// TIA Portal V20 export
FUNCTION "V103" : Void   // FC5, FBD
{ S7_Optimized_Access := 'TRUE' }
// stored: SetENOAutomatically false
   VAR_TEMP
      Temp : "DigVal";
      Temp_1 : "DigVal";
      State : "Service_States";
   END_VAR
BEGIN

REGION Network 1: Channel input
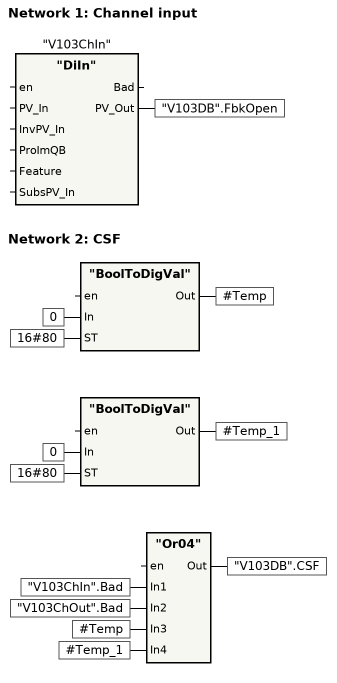
   "V103ChIn"(PV_Out => "V103DB".FbkOpen);   // "DiIn"
END_REGION

REGION Network 2: CSF
   "BoolToDigVal"(In := 0, ST := 16#80, Out => #Temp);
   "BoolToDigVal"(In := 0, ST := 16#80, Out => #Temp_1);
   "Or04"(In1 := "V103ChIn".Bad, In2 := "V103ChOut".Bad, In3 := #Temp, In4 := #Temp_1, Out => "V103DB".CSF);
END_REGION

REGION Network 3: VlvAn Intlock
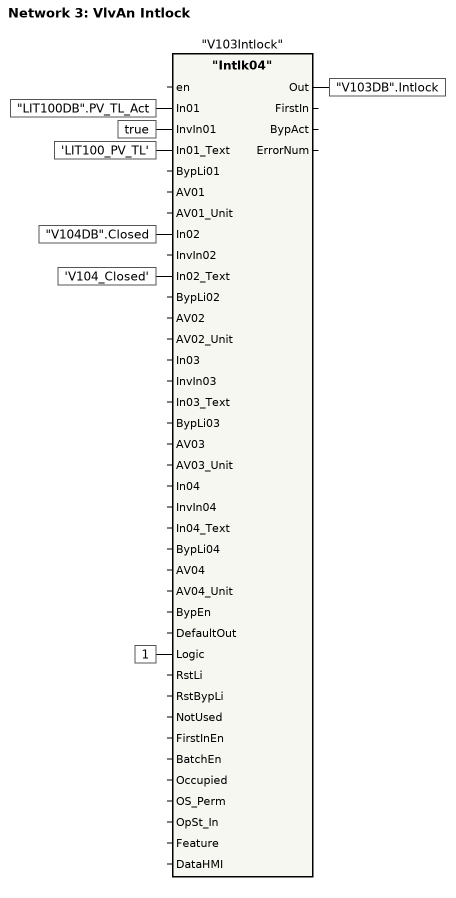
   "V103Intlock"(In01 := "LIT100DB".PV_TL_Act,   // "Intlk04"
                 InvIn01 := true,
                 In01_Text := 'LIT100_PV_TL',
                 In02 := "V104DB".Closed,
                 In02_Text := 'V104_Closed',
                 Logic := 1,
                 Out => "V103DB".Intlock);
END_REGION

REGION Network 4: VlvAnL
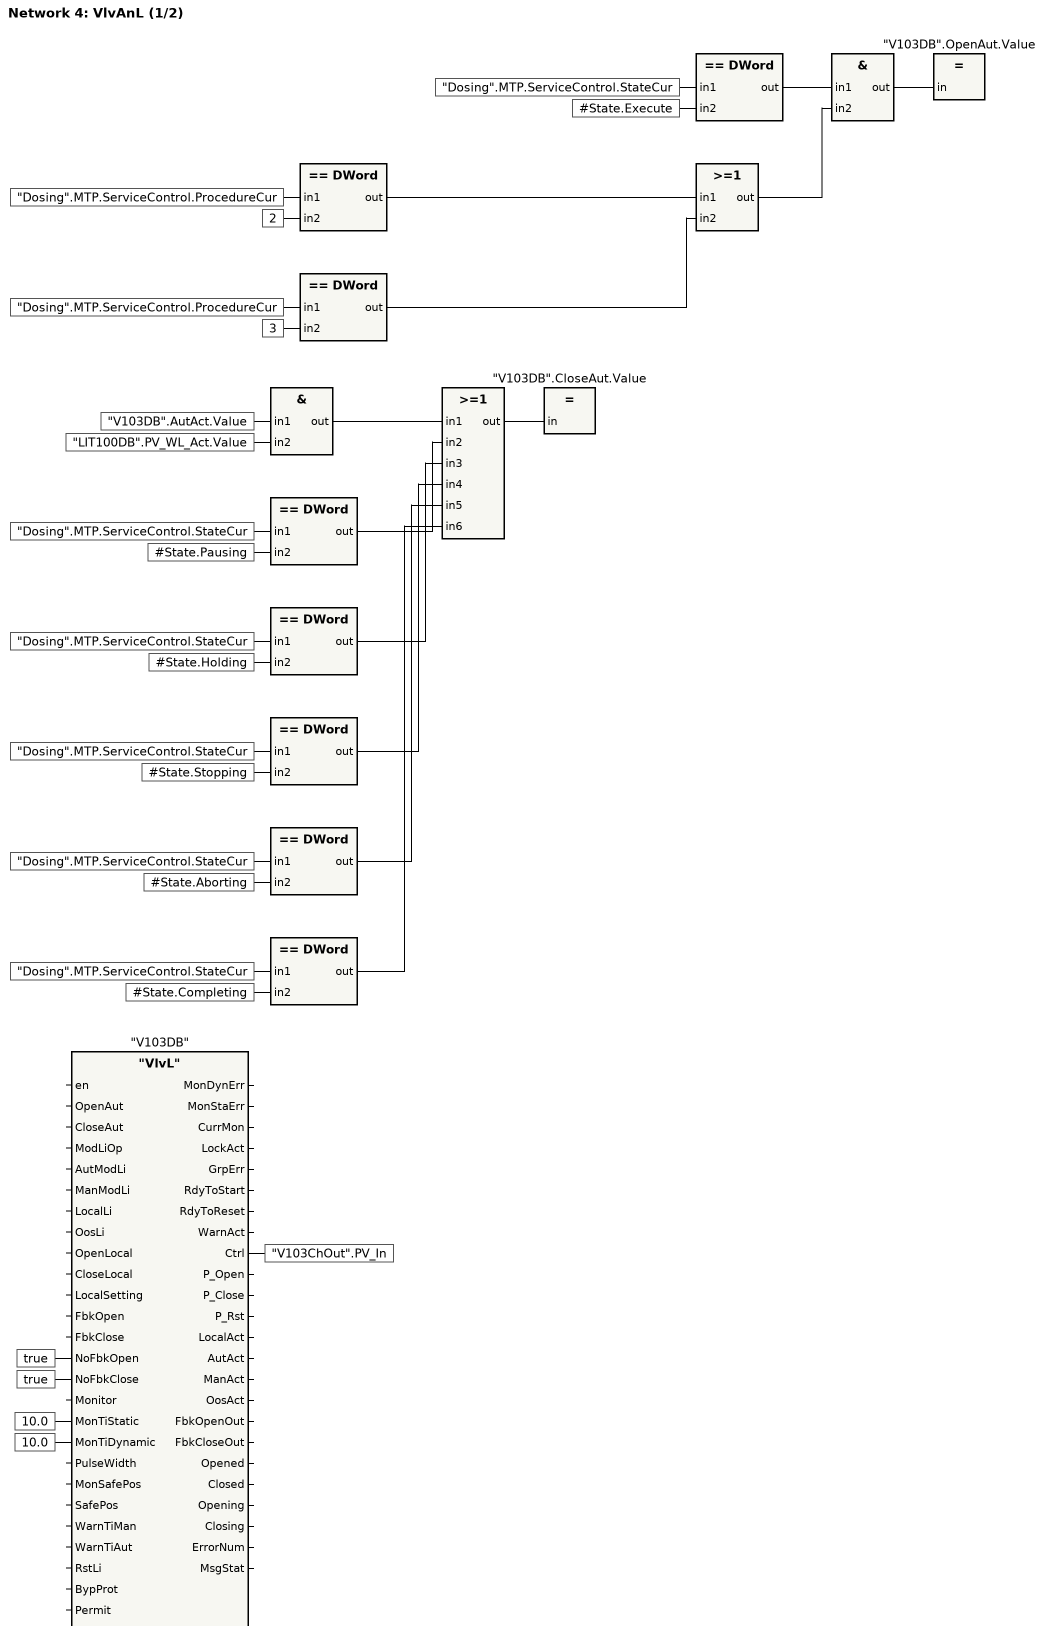
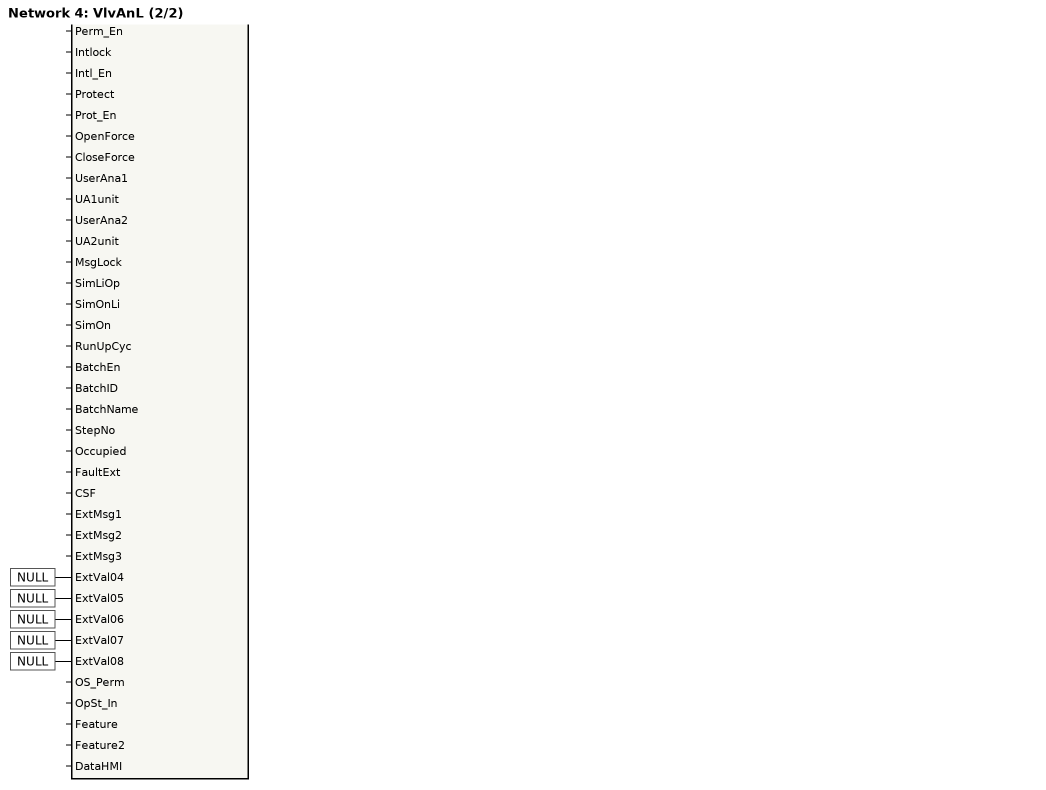
   "V103DB".OpenAut.Value := ("Dosing".MTP.ServiceControl.StateCur = #State.Execute) AND (("Dosing".MTP.ServiceControl.ProcedureCur = 2) OR ("Dosing".MTP.ServiceControl.ProcedureCur = 3));
   "V103DB".CloseAut.Value := ("V103DB".AutAct.Value AND "LIT100DB".PV_WL_Act.Value) OR ("Dosing".MTP.ServiceControl.StateCur = #State.Pausing) OR ("Dosing".MTP.ServiceControl.StateCur = #State.Holding) OR ("Dosing".MTP.ServiceControl.StateCur = #State.Stopping) OR ("Dosing".MTP.ServiceControl.StateCur = #State.Aborting) OR ("Dosing".MTP.ServiceControl.StateCur = #State.Completing);
   "V103DB"(NoFbkOpen := true,   // "VlvL"
            NoFbkClose := true,
            MonTiStatic := 10.0,
            MonTiDynamic := 10.0,
            ExtVal04 := NULL,
            ExtVal05 := NULL,
            ExtVal06 := NULL,
            ExtVal07 := NULL,
            ExtVal08 := NULL,
            Ctrl => "V103ChOut".PV_In);
END_REGION

REGION Network 5: MTP
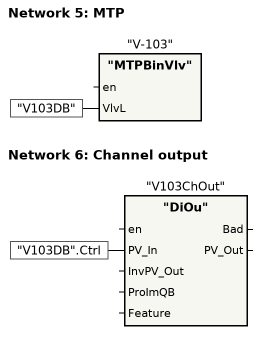
   "V-103"(VlvL := "V103DB");   // "MTPBinVlv"
END_REGION

REGION Network 6: Channel output
   "V103ChOut"(PV_In := "V103DB".Ctrl);   // "DiOu"
END_REGION
END_FUNCTION
